(* IEC 61131-3 sources: axftcmlib/src, 8 files *)

(* ---- ColorSensor.st ---- *)
NAMESPACE Simatic.Ax.axftcmlib

    ///Contains all Colors that the Sensor should know -> Can be expanded
    TYPE
        Colors : INT (UNKNOWN := 10, WHITE := 1, RED := 2,  BLUE := 3); //defaultvalue = UNKNOWN
    END_TYPE

    ///Defines the area in which the values equals a certain color
    TYPE
        ColorRange : STRUCT
            StartValue : INT;
            EndValue : INT;
            Color : colors;
        END_STRUCT;
    END_TYPE

    ///Based on the analogous sensor used in the Fischertechnik FactorySimulation
    CLASS ColorSensor
        VAR PROTECTED
            ColorDetected : BOOL;
        END_VAR

        ///Compares detected value with an array of predefined colorvalues to determin the color
        METHOD PUBLIC detectColor : INT
        VAR_INPUT
        DetectedColorValue : INT;
        ColorArray : ARRAY[*] OF ColorRange;
        END_VAR

        VAR
            Counter : DINT;
        END_VAR
        ColorDetected := FALSE;
        FOR Counter := LOWER_BOUND(ColorArray,1) TO UPPER_BOUND(ColorArray,1) DO
            IF DetectedColorValue >= ColorArray[counter]. StartValue AND DetectedColorValue <= ColorArray[counter].EndValue THEN
                detectColor := ColorArray[Counter].color;
                ColorDetected := TRUE;
            END_IF;
        END_FOR;

            IF ColorDetected = FALSE THEN
                detectColor := Colors#Unknown;
            END_IF;

        END_METHOD

    END_CLASS

END_NAMESPACE

(* ---- IEnablingCm.st ---- *)
///Interface for a class compressor
///contains the basic functions neede for the Fischertechnik models
/// Is used to power a pneumatic cylinder
USING Simatic.Ax.Commands;

NAMESPACE Simatic.Ax.axftcmlib
INTERFACE IEnablingCm
        ///turns the compressor on
        METHOD Enable : itfCommand
        END_METHOD

        ///turns the compressor off
        METHOD Disable : itfCommand
        END_METHOD
    END_INTERFACE

END_NAMESPACE

(* ---- itfCyclicExecution.st ---- *)
NAMESPACE Simatic.Ax.axftcmlib
    INTERFACE itfCyclicExecution
        METHOD RunCyclic END_METHOD
    END_INTERFACE
END_NAMESPACE

(* ---- ControlModuleAbstract.st ---- *)
NAMESPACE Simatic.Ax.axftcmlib
    ///Provides basic functionality for programming on a plc
    /// has acces to the protected Methods and "Contructors" of the classes
    CLASS ABSTRACT ControlModuleAbstract
        VAR PUBLIC

        END_VAR
        VAR PROTECTED
            _init : BOOL;
        END_VAR

        METHOD PUBLIC RunCyclic
            IF (NOT _init) THEN
                THIS._constructor();
                _init := TRUE;
            END_IF;
           THIS._runCyclicCustom();
            ;
        END_METHOD

        METHOD PROTECTED ABSTRACT _runCyclicCustom

        END_METHOD

        METHOD PROTECTED ABSTRACT _constructor

        END_METHOD
    END_CLASS

END_NAMESPACE

(* ---- EnableControlModuleAbstract.st ---- *)
USING Simatic.Ax.Commands;

NAMESPACE Simatic.Ax.axftcmlib
    ///Provides basic functionality for programming on a plc
    /// has acces to the protected Methods and "Contructors" of the classes
    CLASS ABSTRACT EnableControlModuleAbstract EXTENDS Command
        VAR PUBLIC

        END_VAR
        VAR PROTECTED
            _init : BOOL;
            _hasError : BOOL;
            _errorState : WORD;
            _exec : BOOL;
        END_VAR

        METHOD PROTECTED OVERRIDE Execute
            IF (NOT _init) THEN
                THIS._initmethod();
                _init := TRUE;
            END_IF;
           THIS._executeCustom();
            ;
        END_METHOD

        METHOD PROTECTED ABSTRACT _executeCustom

        END_METHOD

        METHOD PROTECTED ABSTRACT _initmethod

        END_METHOD

        METHOD PUBLIC GetErrorStatus : WORD
            GetErrorStatus := _errorState;
        END_METHOD

    END_CLASS

END_NAMESPACE

(* ---- EnablingControlModuleAbstract.st ---- *)
USING Simatic.Ax.Commands;

NAMESPACE Simatic.Ax.axftcmlib
    ///Provides basic functionality for programming on a plc
    /// has acces to the protected Methods and "Contructors" of the classes
    CLASS ABSTRACT EnablingControlModuleAbstract EXTENDS Command
        VAR PUBLIC

        END_VAR
        VAR PROTECTED
            _init : BOOL;
            _hasError : BOOL;
            _errorState : WORD;
            _exec : BOOL;
        END_VAR

        METHOD PROTECTED OVERRIDE Execute
            IF (NOT _init) THEN
                THIS._initmethod();
                _init := TRUE;
            END_IF;
           THIS._executeCustom();
            ;
        END_METHOD

        METHOD PROTECTED ABSTRACT _executeCustom

        END_METHOD

        METHOD PROTECTED ABSTRACT _initmethod

        END_METHOD

        METHOD PUBLIC GetErrorStatus : WORD
            GetErrorStatus := _errorState;
        END_METHOD

    END_CLASS

END_NAMESPACE

(* ---- myClass.st ---- *)
NAMESPACE Simatic.Ax.Library

    {axcode:docs-v0:@simatic-ax/axftcmdlib:MyClass.md}
    CLASS MyClass

        VAR PUBLIC
        END_VAR

        VAR
        END_VAR

        /// Inline Comment for MyMethod. It will be shown, when you hover over the method
        /// This method has no parameters and no return value
        METHOD PUBLIC MyMethod
            ;
        END_METHOD

    END_CLASS

END_NAMESPACE

(* ---- StartGuard.st ---- *)
USING Simatic.Ax.StateFramework;

NAMESPACE Simatic.Ax.axftcmlib

    CLASS StartGuard IMPLEMENTS IGuard

        VAR
            _isStarted : BOOL;
        END_VAR

        METHOD PUBLIC Check : BOOL
            Check := _isStarted;
        END_METHOD

        METHOD PUBLIC Reset
            _isStarted := FALSE;
        END_METHOD

        METHOD PUBLIC Start
            _isStarted := TRUE;
        END_METHOD
    END_CLASS

END_NAMESPACE
